FUNCTION sMsg_Process_Queue : BOOL
VAR_IN_OUT
    pBuffer   : ST_Msg_Buffer;
END_VAR
VAR
    str       			:STRING;
    index     			:UDINT;
	temp_buff			:STRING(4000);
	msg_len				:UDINT;
	free_space			:UDINT;
END_VAR

free_space := 4000 - LEN2(ADR(pBuffer.Pending));

//When there is data to work with and more than 10% free space, spin.
WHILE (pBuffer.MsgQ.Queue.Position[IDX1].HasData) AND (free_space > 400) DO
	// now make sure the new message will fit into whatever remaining space is in the pending buffer
	msg_len := LEN2(ADR(pBuffer.MsgQ.Queue.Position[IDX1].BufferString));
	free_space := 4000 - LEN2(ADR(pBuffer.Pending));
	
	IF msg_len < free_space THEN
		
		concat2(ADR(pBuffer.Pending), ADR(pBuffer.MsgQ.Queue.Position[IDX1].BufferString), ADR(pBuffer.Pending), SIZEOF(pBuffer.Pending));
		
		//cycle the stack
		pBuffer.MsgQ.QueueWorker.ShiftPositionArray(1);
	ELSE
		free_space := 0;
	END_IF
END_WHILE

END_FUNCTION

(* stored: Version 1.1.0.1, ProductVersion 3.1.4024.9
   POU sMsg_Process_Queue: Id {7d194d20-389a-4c1b-90a1-7b948162beef}, SpecialFunc None *)
